// TwinCAT 3 PLC project REST
// ProgramVersion: 3.1.4023.0
// libraries:
//   Tc2_Standard, * (Beckhoff Automation GmbH)
//   Tc2_System, * (Beckhoff Automation GmbH)
//   Tc2_Utilities, * (Beckhoff Automation GmbH)
//   Tc3_IotBase, * (Beckhoff Automation GmbH)
//   Tc3_IotCommunicator, * (Beckhoff Automation GmbH)
//   Tc3_JsonXml, * (Beckhoff Automation GmbH)
//   Tc3_Module, * (Beckhoff Automation GmbH)
// project tree:
//   DUTs/Communicator/ Appdata.TcDUT, ST_SampleData.TcDUT, ST_SampleData_Nested.TcDUT
//   DUTs/ HusetsElfoerbrukning.TcDUT, ST_timData.TcDUT, ST_elpriserTimme.TcDUT, ST_elpriserJustNu24Timmar.TcDUT, parameters.TcDUT, SmartMeterValues.TcDUT, ST_SMHITimeseries.TcDUT, ST_vaederdata.TcDUT, ST_systemtid.TcDUT
//   GVLs/ GVL.TcGVL
//   / PlcTask.TcTTO
//   POUs/GET/ AppCommunicator.TcPOU, BraAttHa.TcPOU, FB_HTTP_Get_SmartMeter.TcPOU, FB_HTTP_Get_Elpris.TcPOU, FB_HTTP_Get_Huset.TcPOU, FB_HTTP_Get_SMHI.TcPOU
//   POUs/ MAIN.TcPOU
// real-time tasks:
//   TASK PlcTask: cycle T#10ms, priority 20, ADS port 350
//   TASK PlcTask1: cycle T#10ms, priority 21, ADS port 351
//   TASK PlcTask2: cycle T#10ms, priority 22, ADS port 352
//   TASK PlcTask3: cycle T#10ms, priority 23, ADS port 353

CONFIGURATION REST
    RESOURCE PLC ON TwinCAT3
        TASK PlcTask(INTERVAL := T#10ms, PRIORITY := 21);
        PROGRAM MAIN WITH PlcTask : MAIN;
    END_RESOURCE
END_CONFIGURATION

// ---- DUTs/Communicator/Appdata.TcDUT
TYPE Appdata :
STRUCT
		
END_STRUCT
	
END_TYPE

// ---- DUTs/Communicator/ST_SampleData.TcDUT
TYPE ST_SampleData :
STRUCT
	{attribute 'iot.DisplayName' := 'Sample STRING on First Level Struct'}
	sSampleString : STRING := 'Sample String';
	
	{attribute 'iot.DisplayName' := 'Sample BOOL on First Level Struct'}
	{attribute 'iot.ReadOnly' := 'true'}
	bSampleBool : BOOL := TRUE;
	
	{attribute 'iot.DisplayName' := 'Sample INT on First Level Struct'}
	{attribute 'iot.Unit' := '%'}
	{attribute 'iot.MinValue' := '0'}
	{attribute 'iot.MaxValue' := '100'}
	{attribute 'iot.ReadOnly' := 'true'}
	iSampleInt : INT := 55;
	
	{attribute 'iot.NestedStructIcon' := 'Room'}
	{attribute 'iot.DisplayName' := 'Second Level Struct'}
	stNestedData : ST_SampleData_Nested;
END_STRUCT
END_TYPE

// ---- DUTs/Communicator/ST_SampleData_Nested.TcDUT
TYPE ST_SampleData_Nested :
STRUCT
	{attribute 'iot.DisplayName' := 'Sample STRING on Second Level Struct'}
	{attribute 'iot.ReadOnly' := 'true'}
	sSampleString : STRING := 'Sample String';
	
	{attribute 'iot.DisplayName' := 'Sample BOOL on Second Level Struct'}
	bSampleBool : BOOL := TRUE;
	
	{attribute 'iot.DisplayName' := 'Sample LREAL on Second Level Struct'}
	{attribute 'iot.Unit' := '°C'}
	{attribute 'iot.ReadOnly' := 'true'}
	{attribute 'iot.DecimalPrecision' := '1'}
	iSampleInt : LREAL := 22.321;
END_STRUCT
END_TYPE

// ---- DUTs/HusetsElfoerbrukning.TcDUT
TYPE HusetsElfoerbrukning :
STRUCT
	power:REAL;
	pf:REAL;
	current:REAL;
	voltage:REAL;
	is_valid:BOOL;
	total:REAL;
	total_returned:REAL;
END_STRUCT
END_TYPE

// ---- DUTs/ST_timData.TcDUT
TYPE ST_timData :
STRUCT
	{attribute 'iot.DisplayName' := 'Timme'}
	DatumTid	: DT;		
	{attribute 'iot.DisplayName' := 'Pris'}
	{attribute 'iot.DecimalPrecision' := '2'}
	{attribute 'iot.Unit' := 'kr'}
	timPris		:	REAL;	//inklusive moms

//Energi
{attribute 'iot.DisplayName' := 'Netto energi'}
	{attribute 'iot.DecimalPrecision' := '2'}
	{attribute 'iot.Unit' := 'kWh'}
	nettoEnergi	: REAL;	//kWh
{attribute 'iot.DisplayName' := 'Såld energi'}
	{attribute 'iot.DecimalPrecision' := '2'}
	{attribute 'iot.Unit' := 'kWh'}
	saaldEnergi	: REAL;	//kWh
{attribute 'iot.DisplayName' := 'Köpt energi'}
	{attribute 'iot.DecimalPrecision' := '2'}
	{attribute 'iot.Unit' := 'kWh'}
	KoeptEnergi	: REAL; //kWh
{attribute 'iot.DisplayName' := 'Husets energi'}
	{attribute 'iot.DecimalPrecision' := '2'}
	{attribute 'iot.Unit' := 'kWh'}
	HusetEnergi : REAL; //kWh

//Effekt 
{attribute 'iot.DisplayName' := 'Topp nettoeffekt'}
	{attribute 'iot.DecimalPrecision' := '2'}
	{attribute 'iot.Unit' := 'W'}
	toppNettoEffekt	: 		REAL:= -10000 ;//W
	{attribute 'iot.DisplayName' := 'Lägsta nettoeffekt'}
	{attribute 'iot.DecimalPrecision' := '2'}
	{attribute 'iot.Unit' := 'W'}
	laegstaNettoEffekt: 	REAL:=10000 ;//W
	{attribute 'iot.DisplayName' := 'Lägsta soleffekt'}
	{attribute 'iot.DecimalPrecision' := '2'}
	{attribute 'iot.Unit' := 'W'}
	leagstaSolEffekt:	REAL:=10000 ;//W
	{attribute 'iot.DisplayName' := 'Högsta soleffekt'}
	{attribute 'iot.DecimalPrecision' := '2'}
	{attribute 'iot.Unit' := 'W'}
	hoegstaSolEffekt:	REAL:= -10000 ;//W
	{attribute 'iot.DisplayName' := 'Lägsta huseffekt'}
	{attribute 'iot.DecimalPrecision' := '2'}
	{attribute 'iot.Unit' := 'W'}
	leagstaHusEffekt:	REAL	:=10000 ;//W
	{attribute 'iot.DisplayName' := 'Högsta huseffekt'}
	{attribute 'iot.DecimalPrecision' := '2'}
	{attribute 'iot.Unit' := 'W'}
	hoegstaHusEffekt:	REAL:= -10000 ;//W

	
//Ekonomi
	{attribute 'iot.DisplayName' := 'Avbetalning solceller'}
	{attribute 'iot.DecimalPrecision' := '2'}
	{attribute 'iot.Unit' := '´kr'}
	avbetalningSolceller	: 	REAL; 	//kr -besparing och såld el
		{attribute 'iot.DisplayName' := 'Sparat solceller'}
	{attribute 'iot.DecimalPrecision' := '2'}
	{attribute 'iot.Unit' := '´kr'}
	sparatSolceller		:	REAL; 	//kr -solel till hushållet
		{attribute 'iot.DisplayName' := 'Sålt'}
	{attribute 'iot.DecimalPrecision' := '2'}
	{attribute 'iot.Unit' := '´kr'}
	saaltSolceller 		: 	REAL; 	//kr -spotpris plus 60 öre skatteavdrag
		{attribute 'iot.DisplayName' := 'Köpt'}
	{attribute 'iot.DecimalPrecision' := '2'}
	{attribute 'iot.Unit' := '´kr'}
	Koept				:	REAL;    //kr 

//Väderdata
	{attribute 'iot.DisplayName' := 'Temperatur'}
	{attribute 'iot.DecimalPrecision' := '2'}
	{attribute 'iot.Unit' := '´°C'}
	Temperatur			:  REAL;    //	°C
		{attribute 'iot.DisplayName' := 'VindGenomsnitt'}
	{attribute 'iot.DecimalPrecision' := '2'}
	{attribute 'iot.Unit' := '´m/s'}
	VindGenomsnitt		: REAL;		// m/s

END_STRUCT
END_TYPE

// ---- DUTs/ST_elpriserTimme.TcDUT
TYPE ST_elpriserTimme :
STRUCT
	SEK_per_kWh: REAL;   //Spotpris kr
    EUR_per_kWh: REAL;   //Spotpris EUR
    EXR: REAL;			//Växelkurs
    time_start: DATE_AND_TIME;
    time_end: DATE_AND_TIME;
END_STRUCT
END_TYPE

// ---- DUTs/ST_elpriserJustNu24Timmar.TcDUT
TYPE ST_elpriserJustNu24Timmar :
STRUCT
	elpriserTimme: ARRAY[1..23] OF ST_elpriserTimme;
	
END_STRUCT
END_TYPE

// ---- DUTs/parameters.TcDUT
TYPE parameters :
STRUCT
END_STRUCT
 parameterArray: ARRAY[0..18] OF ST_vaederdata;
END_TYPE

// ---- DUTs/SmartMeterValues.TcDUT
TYPE SmartMeterValues :
STRUCT
	mac_address: STRING;
	gateway_model: STRING;
	startup_time:  STRING;
    firmware_running: STRING;
    firmware_available: STRING;
    firmware_update_available: STRING;
    wifi_rssi: STRING;
    mqtt_configured: STRING;
    mqtt_server: STRING;
    blynk_configured: STRING;
    Equipment_Id:STRING;
    GasEquipment_Id:STRING;  //ej använd
    ElectricityTariff:STRING;  //ej använd
    EnergyDeliveredTariff1:STRING; //Wh
    EnergyReturnedTariff1: STRING;  //Wh
    EnergyDeliveredTariff2: STRING;  //Wh
    EnergyReturnedTariff2: STRING;  //Wh
    EnergyDelivered: STRING; //Wh
    EnergyReturned: STRING; //Wh
    PowerDelivered_total:STRING; //W   ----- Denna används
    PowerReturned_total: STRING; //W   ----- Denna används
    PowerDelivered_l1: STRING; //W
    PowerDelivered_l2: STRING; //W
    PowerDelivered_l3: STRING; //W
    PowerReturned_l1: STRING; //W
    PowerReturned_l2: STRING; //W
    PowerReturned_l3: STRING; //W
    Voltage_l1: STRING;  //V
    Voltage_l2: STRING; //V
    Voltage_l3: STRING;//V
    Current_l1: STRING; //Amp
    Current_l2: STRING; //Amp
    Current_l3: STRING; //Amp
    GasDelivered: STRING;  //ej använd
    GasDeliveredHour: STRING;  //ej använd
    PowerDeliveredHour: STRING;  //ej använd
    PowerDeliveredNetto: STRING;  //W   ----- Denna används

	
END_STRUCT
END_TYPE

// ---- DUTs/ST_SMHITimeseries.TcDUT
TYPE ST_SMHITimeseries :
STRUCT
	validTime: DATE_AND_TIME;
	parameters: ARRAY[0..18] OF ST_vaederdata;
	
END_STRUCT
END_TYPE

// ---- DUTs/ST_vaederdata.TcDUT
TYPE ST_vaederdata :
STRUCT
	name: STRING;
	levelType: STRING;
	level: REAL;
	unit: STRING;
	values: ARRAY[0..0] OF REAL;
	
END_STRUCT
END_TYPE

// ---- DUTs/ST_systemtid.TcDUT
TYPE ST_systemtid :
STRUCT
	timeLoDW   : UDINT;
    timeHiDW   : UDINT;
END_STRUCT
END_TYPE

// ---- GVLs/GVL.TcGVL
{attribute 'qualified_only'}

VAR_GLOBAL
		HusetsElfoerbrukning: ARRAY[0..23] OF HusetsElfoerbrukning;	
END_VAR
	
VAR_GLOBAL CONSTANT
	//Från EON
	ElOeverfoeringsAvgiftEonKWh: 	REAL:= 0.2645;			// Mars 2023
	EnergiskattKWh: 				REAL:= 0.49;			// Mars 2023
	MomsKWh:		 				REAL:= 0.1886;
	
	NaetNyttaKWh:   REAL:= 0.1663;							// Mars 2023
	
	//Från Kraftringen
	PaaslagMinusRabattKWh: REAL:= 0.009;						// Jan 2023
	//Moms tillkommer också men räknas på spotpriset
	
	//Från Staten
	SkatteAvdragKWh:	REAL:= 0.60;
	
END_VAR

VAR_GLOBAL PERSISTENT
//	timData: ARRAY[0..87600] OF ST_timData;
END_VAR

// ---- POUs/MAIN.TcPOU
PROGRAM MAIN
VAR
	//Communicator
fbCommunicator: AppCommunicator();

	// trigger command execution for Postman-Echo samples
		bGet10sek, bGet24h,bGetSMHI	: BOOL;

	fbHttpClientEonMaetare			: FB_IotHttpClient :=(sHostName:='connectix_smartmeter.local',   // 192.168.68.61
								  	bKeepAlive:=TRUE, tConnectionTimeout:=T#20S);
									
	fbHttpClientHuset			: FB_IotHttpClient :=(sHostName:='192.168.68.200', //Husets El - Shelly
								  	bKeepAlive:=TRUE, tConnectionTimeout:=T#10S);
		
	fbHttpClientElpriset			: FB_IotHttpClient :=(sHostName:='elprisetjustnu.se',
									  	bKeepAlive:=TRUE, tConnectionTimeout:=T#4S);
									
	fbHttpClientSMHI			: FB_IotHttpClient :=(sHostName:='opendata-download-metfcst.smhi.se',
								  	bKeepAlive:=FALSE, tConnectionTimeout:=T#10S);

	fbHttpGetEonMaetare			: FB_HTTP_Get_SmartMeter;
	fbHttpGetHuset				: FB_HTTP_Get_Huset;
	fbHttpGetElpriset			: FB_HTTP_Get_Elpris;
	fbHttpGetSMHI				: FB_HTTP_Get_SMHI;
	



	samladataIntervall: TON;
		
	
	trigger: BOOL;
	loggadata: BOOL;
	raeknartid: TIME;

	nisse: UINT;
	klar: BOOL;
	funkar: BOOL;
	upptagen: BOOL;
	
			systemtid: DT;
	fbGetsytstemtime: GETSYSTEMTIME;
	filetime: T_FILETIME;

	// Tider

	fbLocalTime     : FB_LocalSystemTime;
		systemtidDT: DATE_AND_TIME;
			datumTimmeString: STRING(255);
		datumTimmeDT: DATE_AND_TIME;

	timme: INT;
	TIMEvaerde: TIME;
	TODvaerde: TIME_OF_DAY;
	stringTid: STRING;
	stringTimme: STRING(255);
	timmeloggad: INT;

	stringDatum: STRING(255);
	stringDatumTid: STRING;
	

	bBusyHuset: BOOL;
	bBusyEon: BOOL;
	
	RisingEdge			: R_TRIG;
	nettoEffektW: 			REAL;	//W. Till nätet blir minus och plus från nätet
	husEffektW: 			REAL;	//W
	solEffektW: 			REAL;	//W
	sparadEffektW: 			REAL;	//W

	fbWritePersistent: FB_WritePersistentData;
	bWritePersistent: BOOL;

	fel: UDINT;
	upptagen2: BOOL;
	bErrorCount: INT;
END_VAR

VAR PERSISTENT
	timIndex: INT;    					 //remanent   //Från 0 till 87000 = 10 år
	timData: ARRAY[0..87600] OF ST_timData;
END_VAR



//Communicator appen
fbCommunicator(timData:=timData,timIndex:=timIndex);

//SmartMeter, hämta data en gång per 10sekunder

// EON-mätare - init client parameters at startup
IF NOT fbHttpClientEonMaetare.bConfigured THEN 
	fbHttpClientEonMaetare.nHostPort:= 82;
END_IF

fbHttpClientEonMaetare.Execute();

// Husets-mätare - init client parameters at startup
IF NOT fbHttpClientHuset.bConfigured THEN 
	fbHttpClientHuset.nHostPort:= 80;
END_IF

fbHttpClientHuset.Execute();

// 10 sekunder - Cyklisk fråga med GET - EON-mätare och Hemma-mätare 

samladataIntervall(IN:=trigger, PT:=  T#5S, Q=>klar ,ET=> raeknartid);
IF samladataIntervall.Q THEN
	nisse:=nisse+1;			
	trigger:=FALSE;	
	bGet10sek:=NOT bGet10sek;
ELSE
		trigger:=TRUE;
END_IF

IF fbHttpClientEonMaetare.bConfigured THEN 
		fbHttpGetEonMaetare(timData:=timData,nettoEffektW:=nettoEffektW,bSend:= bGet10sek, fbClient:=fbHttpClientEonMaetare,timIndex:=timIndex,bBusy=>bBusyEon);
END_IF

//Hemmamätare
IF fbHttpClientHuset.bConfigured THEN 
		fbHttpGetHuset(timData:=timData,bSend:=bGet10sek, fbClient:=fbHttpClientHuset, timIndex:=timIndex,husEffektW:= husEffektW, bBusy=>bBusyHuset);
END_IF

RisingEdge(CLK:= NOT bGet10sek );
IF  RisingEdge.Q THEN
	solEffektW:= husEffektW-nettoEffektW;
	IF solEffektW > husEffektW THEN
		sparadEffektW:=husEffektW;
	ELSIF solEffektW>0 AND solEffektW < husEffektW THEN
		sparadEffektW:=solEffektW;
	ELSIF solEffektW<= 0 THEN
		sparadEffektW:=0;
	ELSE
		bErrorCount:=bErrorCount+1;
		
	END_IF
	
	
				IF timData[timIndex].leagstaSolEffekt> solEffektW THEN
					timData[timIndex].leagstaSolEffekt:= solEffektW;
				ELSIF timData[timIndex].hoegstaSolEffekt< solEffektW THEN
					timData[timIndex].hoegstaSolEffekt:= solEffektW;
				END_IF

	timData[timIndex].timPris:= timData[timIndex].timPris;

	//Räkna ut pengar en gång per sampel (10s)
	timData[timIndex].sparatSolceller:= timData[timIndex].sparatSolceller + sparadEffektW/144000*(timData[timIndex].timPris+GVL.ElOeverfoeringsAvgiftEonKWh+GVL.EnergiskattKWh+GVL.MomsKWh+GVL.PaaslagMinusRabattKWh);
	timData[timIndex].avbetalningSolceller:=timData[timIndex].sparatSolceller+timData[timIndex].saaltSolceller;
END_IF

/////////////////////////////////////////////
//24 timmar - Elpriser 

// init client parameters at startup
IF NOT fbHttpClientElpriset.bConfigured THEN 
	fbHttpClientElpriset.stTLS.sVersion:='tlsv1.3';
END_IF


IF fbHttpClientSMHI.bConfigured THEN 
	fbHttpGetSMHI(bSend:=bGet24h, fbClient:=fbHttpClientSMHI, timIndex:=timIndex, timData:=timData, timData:=timData);
END_IF 


IF fbHttpClientElpriset.bConfigured THEN 
	fbHttpGetElpriset(bSend:=bGet24h, fbClient:=fbHttpClientElpriset, stringDatumTid:=stringDatumTid, timIndex:=timIndex, timData:=timData);	
END_IF 


IF timme= 0 THEN
		bGet24h:= TRUE;
ELSE
		bGet24h:= FALSE;
END_IF


fbHttpClientElpriset.Execute();

/////////////////////////////////////////////
//SMHI

// init client parameters at startup
IF NOT fbHttpClientSMHI.bConfigured THEN 
	fbHttpClientSMHI.nHostPort:= 80;
END_IF
	

fbHttpClientSMHI.Execute();



//Räkna fram nuvarande tid och datum
		fbLocalTime(bEnable := TRUE);
		systemtidDT := SYSTEMTIME_TO_DT(fbLocalTime.systemTime);
	  	stringDatumTid:= DT_TO_STRING(systemtidDT);
		datumTimmeString:= MID(stringDatumTid, 17, 1);
		datumTimmeString:= concat(datumTimmeString,'00');
		datumTimmeDT:= STRING_TO_DT(datumTimmeString);

	//timme
	stringTimme:=MID(stringDatumTid, 2, 15);
	timme:= STRING_TO_INT(stringTimme);




// Logga data en gång i timmen
IF timme <> timmeloggad THEN
	bWritePersistent:= TRUE;
	timmeloggad:=timme;
	timIndex:=timIndex+1;
	
 //Data som skall in i struct
	timData[timIndex].DatumTid:=datumTimmeDT;
	
	//Flytta över accumulerad data från förra timmen
	timData[timIndex].avbetalningSolceller:=timData[timIndex-1].avbetalningSolceller;  //Skall inte nollställas
	timData[timIndex].sparatSolceller:=timData[timIndex-1].sparatSolceller;  //Skall inte nollställas
	timData[timIndex].saaltSolceller:=timData[timIndex-1].saaltSolceller;  //Skall inte nollställas
ELSE
	bWritePersistent:= FALSE;
END_IF

//Skriva persistent en gång i timmen
	fbWritePersistent(START:=bWritePersistent,TMOUT:=DEFAULT_ADS_TIMEOUT,PORT:=851,BUSY=>upptagen2, ERRID=>fel);

	IF upptagen2 THEN
		nisse:=nisse+1;
	END_IF

END_PROGRAM

// ---- POUs/GET/AppCommunicator.TcPOU
FUNCTION_BLOCK AppCommunicator
// This sample defines a simple TwinCAT Iot Device (fbIot), which connects to localhost.
// As soon as connection is established, the timer starts and data (stData) is sent every second.
//
// A message is sent once on startup and can be triggered by setting bSendMessage to TRUE.

VAR_INPUT
		timData: REFERENCE TO ARRAY[0..87600] OF ST_timData;
	timIndex: REFERENCE TO INT;
END_VAR

VAR
	
	// Declare FB_IotCommunicator
	fbIot : FB_IotCommunicator := (sHostName := '127.0.0.1',
									nPort := 1883,
									sMainTopic := 'Husdata',
									sDeviceName := 'Hemma',
									sUser := 'FullSampleUser',
									sPassword := '',
									sDeviceIcon := 'House');

	
	// Trigger send message
	bSendMessage : BOOL := TRUE;
	
	// Timer to send data only once per second
	timer : TON;

END_VAR

// .Execute() has to be called cyclically
// TRUE --> connection will be established
// FALSE --> connection will be closed
fbIot.Execute(TRUE);




// Start timer when fbIot is connected
IF fbIot.bConnected  THEN
	timer(IN := TRUE, PT := T#1000MS);
END_IF

// Send data, if timer is expired
IF timer.Q THEN
	timer(IN := FALSE);
	
	fbIot.SendData(ADR(timData[timIndex]), SIZEOF(timData[timIndex]));
	//fbIot2.SendDataAsString(ADR(sampleString), LEN(sampleString));
END_IF

(*
// Receive variable changes, triggered by app
IF fbIot.fbCommand.bAvailable THEN
	// Receive data for first level struct
	IF fbIot.fbCommand.sVarName = 'sSampleString' THEN
//fbIot.fbCommand.GetValue(ADR(stData), SIZEOF(stData), E_IotCommunicatorDatatype.);
		fbIot.fbCommand.GetValue(ADR(stData.sSampleString), SIZEOF(stData.sSampleString), E_IotCommunicatorDatatype.type_STRING);
	END_IF
	// Receive data for second level struct
	IF fbIot.fbCommand.sVarName = 'stNestedData.bSampleBool' THEN
		fbIot.fbCommand.GetValue(ADR(stData.stNestedData.bSampleBool), SIZEOF(stData.stNestedData.bSampleBool), E_IotCommunicatorDatatype.type_BOOL);
	END_IF
	
	fbIot.SendData(ADR(stData), SIZEOF(stData));
	fbIot.fbCommand.Remove();
END_IF
*)
// Send message, if bSendMessage is set to true
IF bSendMessage THEN
	fbIot.SendMessage('This is a sample message from TF6730_FullSample');

	bSendMessage := FALSE;
END_IF

END_FUNCTION_BLOCK

// ---- POUs/GET/FB_HTTP_Get_SmartMeter.TcPOU
FUNCTION_BLOCK FB_HTTP_Get_SmartMeter
VAR_INPUT
	bSend				: BOOL;
	timData: REFERENCE TO ARRAY[0..87600] OF ST_timData;
	timIndex: REFERENCE TO INT;
	nettoEffektW:REFERENCE TO REAL;
END_VAR
VAR_IN_OUT
	fbClient			: FB_IotHttpClient;
END_VAR
VAR_OUTPUT
	bBusy				: BOOL;
	bError				: BOOL;
END_VAR
VAR
	fbRequest			: FB_IotHttpRequest;
	
		fbJsonDataType	: FB_JsonReadWriteDataType;
		felkod			: HRESULT;			
	pContent: PVOID;
	nState				: UDINT;
	RisingEdge			: R_TRIG;
	
	bGetContentResult	: BOOL;
	sContent			: STRING(1100);
	
	bGetJsonResult		: BOOL;
	
	nReqCount			: UDINT;	
	nResCount			: UDINT;
	nValidResCount		: UDINT;
	nErrCount			: UDINT;


	nisse: REAL;
	stSmartDataMomentan: SmartMeterValues;
	nisse1: REAL;
END_VAR

RisingEdge(CLK:= bSend );



CASE nState OF
0:	
	IF RisingEdge.Q THEN 
		IF fbRequest.SendRequest(sUri:='/smartmeter/api/read', fbClient:=fbClient, eRequestType:=ETcIotHttpRequestType.HTTP_Get, 0, 0, 0) THEN				
		
		nState:= 1;
			nReqCount:= nReqCount+1;
			bBusy:= TRUE;
			bError:= FALSE;
		END_IF				
	END_IF
1:

	IF NOT fbRequest.bBusy THEN
		bError:= TRUE;
		IF NOT fbRequest.bError THEN	
			

			
//Hämta data från mätarens HTTP REST API och lägg i string
			bGetContentResult:= fbRequest.GetContent(pContent:= ADR(sContent), nContentSize:= SIZEOF(sContent), bSetNullTermination:= TRUE);
			
			
			IF fbRequest.nStatusCode >= 200 AND fbRequest.nStatusCode < 300 THEN
				bGetJsonResult:= FALSE;
			
			//Kopiera hela den importerade JSON-formaterade datasträngen och lägg i en motsvarande TwinCAT-struktur
			IF fbJsonDataType.SetSymbolFromJson(sContent, 'SmartMeterValues', SIZEOF(stSmartDataMomentan), ADR(stSmartDataMomentan), hrErrorCode=> felkod) THEN
						bError:= FALSE;
					END_IF	
			
			//räkna ut lägsta och högsta effekt
			IF felkod = 0 THEN
					

				nettoEffektW:= STRING_TO_REAL(stSmartDataMomentan.PowerDeliveredNetto);
				
				
			END_IF	
			
				//skriv in i Struct
				timData[timIndex].nettoEnergi:= timData[timIndex].nettoEnergi+ (nettoEffektW/144000);    //144 sampel per timme
				
				IF nettoEffektW >0 THEN
					timData[timIndex].KoeptEnergi:= timData[timIndex].KoeptEnergi+(nettoEffektW/144000);   //144 sampel per timme
				ELSE
						timData[timIndex].saaldEnergi:= timData[timIndex].saaldEnergi- (nettoEffektW/144000);   //144 sampel per timme
				END_IF
				
				IF timData[timIndex].laegstaNettoEffekt> nettoEffektW THEN 	
					timData[timIndex].laegstaNettoEffekt:=nettoEffektW;
				ELSIF timData[timIndex].toppNettoEffekt< nettoEffektW THEN 	
					timData[timIndex].toppNettoEffekt:=nettoEffektW;			
				END_IF
			
				nResCount:= nResCount+1;			
			END_IF
		END_IF
			nisse:=nisse+1;
		nState:= 2;
		bBusy:= FALSE;
		IF bError THEN
			nErrCount:= nErrCount+1;
		END_IF
	END_IF  	

2:   //Räkna ut pengar
IF nettoEffektW >0 THEN
	timData[timIndex].Koept:= timData[timIndex].Koept + nettoEffektW/144000*(timData[timIndex].timPris+GVL.ElOeverfoeringsAvgiftEonKWh+GVL.EnergiskattKWh+GVL.MomsKWh+GVL.PaaslagMinusRabattKWh);
ELSE
	timData[timIndex].saaltSolceller:= timData[timIndex].saaltSolceller-(nettoEffektW/144000*(timData[timIndex].timPris+GVL.NaetNyttaKWh+GVL.SkatteAvdragKWh));  //Sålt i kr
END_IF


nState:= 0;

	
END_CASE

END_FUNCTION_BLOCK

// ---- POUs/GET/FB_HTTP_Get_Huset.TcPOU
FUNCTION_BLOCK FB_HTTP_Get_Huset
VAR_INPUT
	bSend				: BOOL;
	//timDataMomentan:REFERENCE TO ST_timData;
		timData: REFERENCE TO ARRAY[0..87600] OF ST_timData;
		timIndex: REFERENCE TO INT;
	husEffektW:REFERENCE TO REAL;
END_VAR
VAR_IN_OUT
	fbClient			: FB_IotHttpClient;
END_VAR
VAR_OUTPUT
	bBusy				: BOOL;
	bError				: BOOL;
END_VAR
VAR
	fbRequest			: FB_IotHttpRequest;
	fbJson				: FB_JsonDomParser;
	
		fbJsonDataType	: FB_JsonReadWriteDataType;
		felkod			: HRESULT;			
	pContent: PVOID;
	nState				: UDINT;
	RisingEdge			: R_TRIG;
	
	bGetContentResult	: BOOL;
	sContent			: STRING(1100);
	
	bGetJsonResult		: BOOL;
	jsonDoc				: SJsonValue;
	jsonVal				: SJsonValue;
	sResultValue		: STRING;
	
	nReqCount			: UDINT;	
	nResCount			: UDINT;
	nValidResCount		: UDINT;
	nErrCount			: UDINT;
	Vaerde: LINT;
	
	Effektlaegsta: REAL :=100000.0 ;
	Effekthoegsta: REAL;
	stHusetsDataMomentan: ARRAY[0..2] OF HusetsElfoerbrukning;

	Funkar: BOOL;
	nisse: INT;

	i: INT;
	nStateMAx: UDINT;
	
	
	nState1: UDINT;
	nState2: UDINT;
	nState3: UDINT;

END_VAR

RisingEdge(CLK:= bSend );

IF nStateMAx < nState THEN
	nStateMAx := nState;
END_IF

CASE nState OF
	

0:	
	IF RisingEdge.Q THEN 
		IF fbRequest.SendRequest(sUri:='/emeter/0', fbClient:=fbClient, eRequestType:=ETcIotHttpRequestType.HTTP_Get, 0, 0, 0) THEN				
		
		nState:= 1;
			nReqCount:= nReqCount+1;
			bBusy:= TRUE;
			bError:= FALSE;
		END_IF					
	END_IF
1:

	IF NOT fbRequest.bBusy THEN
		bError:= TRUE;
		IF NOT fbRequest.bError THEN	
			////////
			GetContent();
		
		END_IF
			nisse:=nisse+1;
		nState:= 2;                              //Ändra deta
		bBusy:= FALSE;
		IF bError THEN
			nErrCount:= nErrCount+1;
		END_IF
	END_IF  

	

	
2:	
	//IF RisingEdge.Q THEN 
	IF NOT fbRequest.bBusy THEN
		IF fbRequest.SendRequest(sUri:='/emeter/1', fbClient:=fbClient, eRequestType:=ETcIotHttpRequestType.HTTP_Get, 0, 0, 0) THEN				
		
		nState:= 3;
			nReqCount:= nReqCount+1;
			bBusy:= TRUE;
			bError:= FALSE;
		END_IF		
	END_IF			
	//END_IF
3:


IF NOT fbRequest.bBusy THEN
		bError:= TRUE;
		IF NOT fbRequest.bError THEN	
			////////
			GetContent();
		
		END_IF
			nisse:=nisse+1;
		nState:= 4;                              
		bBusy:= FALSE;
		IF bError THEN
			nErrCount:= nErrCount+1;
		END_IF
	END_IF  

	
	
	4:	
		//IF RisingEdge.Q THEN 
	IF NOT fbRequest.bBusy THEN
		IF fbRequest.SendRequest(sUri:='/emeter/2', fbClient:=fbClient, eRequestType:=ETcIotHttpRequestType.HTTP_Get, 0, 0, 0) THEN				
		
		nState:= 5;
			nReqCount:= nReqCount+1;
			bBusy:= TRUE;
			bError:= FALSE;
		END_IF		
	END_IF			
	//END_IF
5:

	
IF NOT fbRequest.bBusy THEN
		bError:= TRUE;
		IF NOT fbRequest.bError THEN	
			////////
			GetContent();
		
		END_IF
			nisse:=nisse+1;
		nState:= 6;                              
		bBusy:= FALSE;
		IF bError THEN
			nErrCount:= nErrCount+1;
		END_IF
	END_IF  

6:   //Räkna ut pengar
	//HusetsEffekt+timDataMomentan.Koept
//timDataMomentan.nettoEnergi

nState:= 0;

	
END_CASE

METHOD GetContent : BOOL
VAR_INPUT
END_VAR

VAR

	n: INT;

	
END_VAR
//Hämta data från mätarens HTTP REST API och lägg i string
			bGetContentResult:= fbRequest.GetContent(pContent:= ADR(sContent), nContentSize:= SIZEOF(sContent), bSetNullTermination:= TRUE);
						
			IF fbRequest.nStatusCode >= 200 AND fbRequest.nStatusCode < 300 THEN
				bGetJsonResult:= FALSE;
			
			//Kopiera hela den importerade JSON-formaterade datasträngen och lägg i en motsvarande TwinCAT-struktur
			IF fbJsonDataType.SetSymbolFromJson(sContent, 'HusetsElfoerbrukning', SIZEOF(stHusetsDataMomentan[(nState-1)/2]), ADR(stHusetsDataMomentan[(nState-1)/2]), hrErrorCode=> felkod) THEN
						bError:= FALSE;
			END_IF	
			
				
				//När alla faser är genomgångna								
				IF nState = 5 THEN
				
				husEffektW :=0;	
				FOR n :=0 TO 2 DO
						timData[timIndex].HusetEnergi:= timData[timIndex].HusetEnergi+ (stHusetsDataMomentan[n].power/144000);		//Accumulerad Energi, nollställs varje timme
						husEffektW := husEffektW+ stHusetsDataMomentan[n].power;					//tillfällig effekt
	
						
					END_FOR
						//skriv in i Struct				
					IF timData[timIndex].leagstaHusEffekt> husEffektW THEN 	
					timData[timIndex].leagstaHusEffekt:=husEffektW;
					END_IF
				
					IF timData[timIndex].hoegstaHusEffekt< husEffektW  THEN 	
					timData[timIndex].hoegstaHusEffekt:= husEffektW;
					END_IF
					
					
				END_IF
			
		
				nResCount:= nResCount+1;			
			END_IF
END_METHOD

END_FUNCTION_BLOCK

// ---- POUs/GET/FB_HTTP_Get_Elpris.TcPOU
FUNCTION_BLOCK FB_HTTP_Get_Elpris
VAR_INPUT
	bSend			: BOOL;
	//:REFERENCE TO ST_timData;
	timData: REFERENCE TO ARRAY[0..87600] OF ST_timData;
	stringDatumTid: STRING;
	timIndex: REFERENCE TO INT;
END_VAR
VAR_IN_OUT
	fbClient			: FB_IotHttpClient;
END_VAR
VAR_OUTPUT
	bBusy				: BOOL;
	bError				: BOOL;
END_VAR
VAR
		elpriserTimme: ARRAY[0..23] OF ST_elpriserTimme; //från elpriserjustnu.se
	fbRequest			: FB_IotHttpRequest;

	fbJson				: FB_JsonDomParser;
	
		fbJsonDataType	: FB_JsonReadWriteDataType;
		felkod			: HRESULT;			
	pContent: PVOID;
	nState				: UDINT;
	RisingEdge			: R_TRIG;
	
	bGetContentResult	: BOOL;
	sContent			: STRING(5000);
	
	bGetJsonResult		: BOOL;
	jsonDoc				: SJsonValue;
	jsonVal				: SJsonValue;
	sResultValue		: STRING;
	
	nReqCount			: UDINT;	
	nResCount			: UDINT;
	nValidResCount		: UDINT;
	nErrCount			: UDINT;
	Vaerde: LINT;
	Energi: REAL;
	Energilaegsta: REAL :=100000.0 ;
	Energihoegsta: REAL;
	n: INT;
	Funkar: BOOL;
	nisse: INT;
	kod1: UINT;
	kod2: UINT;
	Location: STRING(200);
	
	
	storlek: UINT;
	storleken: UDINT;
	nIndex: UDINT;
	nSize: UDINT;
	sJsonArrayIndex: Sjsonvalue;
	
	sJsonArray			:SJsonValue;

	SCopiedJson: STRING(200);

	
	sUri: STRING(255);
	stringDatum: STRING(255);
	stringAar: STRING(255);
	i: INT;
	nisses: REAL;
	kalle: INT;
	sldg: REAL;
	bTestRef1: BOOL;
END_VAR

RisingEdge(CLK:= bSend );


CASE nState OF
0:	
	IF RisingEdge.Q THEN 
	kalle:=kalle+1;
		 
			stringAar:=MID(stringDatumTid, 4, 4);
				stringDatum:=MID(stringDatumTid, 5, 9);
			 
			 sUri:=concat('/api/v1/prices/', stringAar);
			 sUri:=concat(sUri,'/'); 
			 sUri:=concat(sUri,stringDatum);
			 sUri:=concat(sUri,'_SE4.json');
			 //sUri:='/api/v1/prices/2023/02-14_SE4.json'

		IF fbRequest.SendRequest(sUri:=sUri, fbClient:=fbClient, eRequestType:=ETcIotHttpRequestType.HTTP_GET, 0, 0, 0) THEN
			
			nState:= 1;
			nReqCount:= nReqCount+1;
			bBusy:= TRUE;
			bError:= FALSE;
			sUri:='';
		END_IF					
	END_IF
1:
	IF NOT fbRequest.bBusy THEN
		nisse:=nisse+1;
			fbRequest.GetHeaderField(sField:='Location',pValue:=ADR(Location),nValueSize:= SIZEOF(Location));
		kod1:=fbRequest.nStatusCode;
		bError:= TRUE;
		IF NOT fbRequest.bError THEN	
			//Hämta data och lägg i string
		
		
		
			bGetContentResult:= fbRequest.GetContent(pContent:= ADR(sContent), nContentSize:= SIZEOF(sContent), bSetNullTermination:= TRUE);
		
			storleken:=fbRequest.nContentSize;
			
			IF fbRequest.nStatusCode >= 200 AND fbRequest.nStatusCode < 300 THEN
				bGetJsonResult:= FALSE;
				jsonDoc:= fbRequest.GetJsonDomContent(fbJson);
				IF jsonDoc <> 0 THEN
					bGetJsonResult:= TRUE;
					
					//sJsonArray:=fbJson.FindMember(jsonDoc, 'timeSeries');
				
					nSize:= LIMIT(1, fbJson.GetArraySize(jsonDoc), 100);
					
					FOR nIndex:= 0 TO (nSize-1) DO   //Alltid 0-23 timmar
						sJsonArrayIndex:= fbJson.GetArrayValueByIdx(jsonDoc, nIndex);
						fbJson.CopyJson(sJsonArrayIndex, SCopiedJson, SIZEOF(SCopiedJson));
						fbJsonDataType.SetSymbolFromJson(sCopiedJson, 'ST_elpriserTimme', SIZEOF(elpriserTimme[nIndex]), ADR(elpriserTimme[nIndex]));
					END_FOR
			(*	
				//Kopiera hela den importerade JSON-formaterade datasträngen och lägg i en motsvarande TwinCAT-struktur
				IF fbJsonDataType.SetSymbolFromJson(sContent, 'ST_elpriserJustNu24Timmar', SIZEOF(elpriserTimme), ADR(elpriserTimme), hrErrorCode=> felkod) THEN
						bError:= FALSE;
				END_IF	
		*)
		
		//Stoppa in dygnets elpriser

		
FOR i:= 0 TO (23) DO
	timData[timIndex+i].timPris:= elpriserTimme[i].SEK_per_kWh;
	//sldg:= elpriserTimme[i].SEK_per_kWh;
END_FOR

				nResCount:= nResCount+1 ;	
				

			END_IF
		END_IF
		nState:= 0;
		bBusy:= FALSE;
		IF bError THEN
			nErrCount:= nErrCount+1;
		END_IF
	END_IF  
END_IF	


END_CASE

END_FUNCTION_BLOCK

// ---- POUs/GET/FB_HTTP_Get_SMHI.TcPOU
FUNCTION_BLOCK FB_HTTP_Get_SMHI
VAR_INPUT
	bSend				: BOOL;
	//timDataMomentan:REFERENCE TO ST_timData;
	timData: REFERENCE TO ARRAY[0..87600] OF ST_timData;
	timIndex: REFERENCE TO INT;
END_VAR
VAR_IN_OUT
	fbClient			: FB_IotHttpClient;
END_VAR
VAR_OUTPUT
	bBusy				: BOOL;
	bError				: BOOL;
END_VAR
VAR
	
	fbRequest			: FB_IotHttpRequest;
	;
	fbJson				: FB_JsonDomParser;

		fbJsonDataType	: FB_JsonReadWriteDataType;
		felkod			: HRESULT;			
	pContent: PVOID;
	nState				: UDINT;
	RisingEdge			: R_TRIG;
	
	bGetContentResult	: BOOL;
	sContent			: STRING(150000);
	
	bGetJsonResult		: BOOL;
	jsonDoc				: SJsonValue;
	jsonVal				: SJsonValue;
	sJsonArray			:SJsonValue;
	sJsonArrayIndex		: SJsonValue;
	
	sResultValue		: STRING;
	
	nReqCount			: UDINT;	
	nResCount			: UDINT;
	nValidResCount		: UDINT;
	nErrCount			: UDINT;
	Vaerde: LINT;
	Energi: REAL;
	Energilaegsta: REAL :=100000.0 ;
	Energihoegsta: REAL;
	n: INT;
	Funkar: BOOL;
	nisse: UDINT;
	nSize: UDINT;
	i: INT;
	
	nIndex: UDINT;
	SCopiedJson: STRING(6000);
	storlek: UINT;
	p: INT;
	
	timeseries: ARRAY[0..100] OF ST_SMHITimeseries;
END_VAR

RisingEdge(CLK:= bSend );
CASE nState OF
0:	
	IF RisingEdge.Q THEN 
		//hämtar väderdata för Glumslöv
		IF Funkar:= fbRequest.SendRequest(sUri:='/api/category/pmp3g/version/2/geotype/point/lon/12.809493/lat/55.937773/data.json', fbClient:=fbClient, eRequestType:=ETcIotHttpRequestType.HTTP_GET, 0, 0, 0) THEN				

		nState:= 1;
			nReqCount:= nReqCount+1;
			bBusy:= TRUE;
			bError:= FALSE;
		END_IF					
	END_IF
1:
	IF NOT fbRequest.bBusy THEN
		bError:= TRUE;
		IF NOT fbRequest.bError THEN	
		bGetContentResult:= fbRequest.GetContent(pContent:= ADR(sContent), nContentSize:= SIZEOF(sContent), bSetNullTermination:= TRUE);
		nisse:= fbRequest.nContentSize;
		
			IF fbRequest.nStatusCode >= 200 AND fbRequest.nStatusCode < 300 THEN
				bGetJsonResult:= FALSE;
				jsonDoc:= fbRequest.GetJsonDomContent(fbJson);
				IF jsonDoc <> 0 THEN
					bGetJsonResult:= TRUE;
					
					sJsonArray:=fbJson.FindMember(jsonDoc, 'timeSeries');
					
					nSize:= LIMIT(1, fbJson.GetArraySize(sJsonArray), 100);
					
					FOR nIndex:= 0 TO (nSize-1) DO
						sJsonArrayIndex:= fbJson.GetArrayValueByIdx(sJsonArray, nIndex);
						fbJson.CopyJson(sJsonArrayIndex, SCopiedJson, SIZEOF(SCopiedJson));
						fbJsonDataType.SetSymbolFromJson(sCopiedJson, 'ST_SMHITimeseries', SIZEOF(timeseries[nIndex]), ADR(timeseries[nIndex]));
												
					END_FOR

				FOR i:=1 TO 24 DO    // timeseries[0] brukar vara kl 23 föregående dygn
					FOR p:=0 TO 18 DO
						IF	timeseries[i].parameters[p].name = 't' THEN
							timData[timIndex+i].Temperatur:= timeseries[i].parameters[p].values[0];
						END_IF
						IF	timeseries[i].parameters[p].name = 'ws' THEN
							timData[timIndex+i].VindGenomsnitt:= timeseries[i].parameters[p].values[0];
						END_IF					
						
						
					END_FOR
				END_FOR
				
					
					
				END_IF	
				nResCount:= nResCount+1;			
			END_IF
		END_IF
		nState:= 0;
		bBusy:= FALSE;
		IF bError THEN
			nErrCount:= nErrCount+1;
		END_IF
	END_IF  	
END_CASE

END_FUNCTION_BLOCK

// ---- POUs/GET/BraAttHa.TcPOU
FUNCTION_BLOCK BraAttHa
VAR_INPUT
	timData: REFERENCE TO ARRAY[0..87600] OF ST_timData;
END_VAR
VAR_OUTPUT
END_VAR
VAR
	eWriteState: (FILE_OPEN_TRIGGER,FILE_OPEN, WAIT_FOR_EVENT, WRITE_EVENT_TRIGGER,WRITE_EVENT, FILE_CLOSE_TRIGGER, FILE_CLOSE, ERROR); //används i CASE istället för siffror
	timestruct             : TIMESTRUCT;    
	fbMeRingBuffer: FB_MemRingBuffer;   //Ringbuffert
	
	//Hämta lokal tid
	   bInit           : BOOL;
    nTime           : UINT;
    tBufferTime     : TIME;
    dtBufferDT      : DT;
    nCalcBuffer     : UDINT;
    sMs             : STRING;
    sLogTime        : STRING;
    sLogTimeWithMs  : STRING;
    stSystemTime    : TIMESTRUCT;
    fbLocalTime     : FB_LocalSystemTime;
	bTestRef1: BOOL;
	nisse: BOOL;
	
	arraydata: ARRAY[0..9] OF ST_elpriserTimme;
END_VAR


//Hämta lokal tid
	fbLocalTime(bEnable := TRUE);
	  dtBufferDT := SYSTEMTIME_TO_DT(fbLocalTime.systemTime);fbLocalTime(bEnable := TRUE);
IF NOT bInit
THEN
    dtBufferDT := SYSTEMTIME_TO_DT(fbLocalTime.systemTime);
    IF fbLocalTime.bValid 
    THEN
        bInit := TRUE;
    END_IF
ELSE
    nTime := nTime + 1;
    tBufferTime := UINT_TO_TIME(nTime*10);
    IF tBufferTime = T#1S
    THEN
        //Add a second to your system time
        ntime := 0;
        nCalcBuffer := DT_TO_UDINT(dtBufferDT)+1;
        dtBufferDT := UDINT_TO_DT(nCalcBuffer);
        sLogTime := DT_TO_STRING(dtBufferDT);
        sLogTimeWithMs := sLogTime;
    ELSE
        //Add ms string time-stamp
        sMs := TIME_TO_STRING(tBufferTime);
        sLogTimeWithMs := CONCAT(sLogTime,sMs);
    END_IF
END_IF

//Kolla om en REFERENCE-variabel är VALID. Är den inte det så kolla om den är med i anropet av FB:t
		bTestRef1  := __ISVALIDREF(timData);
		
		
		IF nisse THEN
	MEMCPY(ADR(arraydata[0]),ADR(arraydata[1]), SIZEOF(arraydata[1])); //Kopiera en hel strukt på en gång. 
 
END_IF

END_FUNCTION_BLOCK
